(* IEC 61131-3 sources: HappyLearnCodesys/content/softmotion/CNC09_ToolLengthCorr, 3 files *)

(* ---- GVL.st ---- *)
VAR_GLOBAL CONSTANT
	gc_dwCycle : DWORD := 4000;
	gc_eOriConvention : SMC_ORI_CONVENTION := SMC_ORI_CONVENTION.ZYZ;
END_VAR

(* ---- CNC.st ---- *)
PROGRAM CNC
VAR
	iState: INT;
	pX, pY, pZ, pA: MC_Power;

	ipo: SMC_Interpolator;
	trafo: SMC_TRAFO_Gantry3;
	trafof: SMC_TRAFOF_Gantry3D;
	cabpX, cabpY, cabpZ, cabpA: SMC_ControlAxisByPos;

	tlc : SMC_ToolLengthCorr;
END_VAR

pX(
	Enable:= TRUE,
	bRegulatorOn:= TRUE,
	bDriveStart:= TRUE,
	Axis:= AxisX);
pY(
	Enable:= TRUE,
	bRegulatorOn:= TRUE,
	bDriveStart:= TRUE,
	Axis:= AxisY);
pZ(
	Enable:= TRUE,
	bRegulatorOn:= TRUE,
	bDriveStart:= TRUE,
	Axis:= AxisZ);
pA(
	Enable:= TRUE,
	bRegulatorOn:= TRUE,
	bDriveStart:= TRUE,
	Axis:= AxisA);

CASE iState OF
0:
	IF pX.Status AND pY.Status AND pZ.Status AND pA.Status THEN
		iState := 100;
	END_IF
100:
	Interpolation();
END_CASE

(* ---- CNC_PreparePath.st ---- *)
PROGRAM CNC_PreparePath
VAR_INPUT
	xStart: BOOL;
	sFileName: STRING := 'Application/CNC.cnc';
END_VAR
VAR_OUTPUT
	xStartIpo: BOOL;
	poqPath: Pointer to SMC_Outqueue;
END_VAR
VAR
	iState: INT;
	rncf2 : SMC_ReadNCFile2;
	nci : SMC_NCInterpreter;
	cv : SMC_CheckVelocities;
	aBufInterpreter : ARRAY[0..99] OF SMC_GeoInfo ;
END_VAR

poqPath := cv.poqDataOut;

CASE iState OF
0:	// idle
	IF xStart THEN
		iState := 10;
		xStartIpo := FALSE;
		rncf2(bExecute:= FALSE);
		nci(bExecute:= FALSE,sentences:= rncf2.sentences);
		cv(bExecute:= FALSE);
		xStart := FALSE;
	END_IF

10:	// start reading and processing
	rncf2(
        bExecute:= TRUE,
		sFileName:= sFileName);

	nci(
        bExecute:= TRUE,
		sentences := rncf2.sentences,
		nSizeOutQueue:= SIZEOF(aBufInterpreter),
		pbyBufferOutQueue:= ADR(aBufInterpreter),
        bEnableSyntaxChecks:= TRUE,
        eOriConv:= gc_eOriConvention);

	cv(
        bExecute:= TRUE,
		poqDataIn:= nci.poqDataOut);

	xStartIpo := TRUE;
	IF NOT cv.bBusy THEN
		iState:=0;
	END_IF
END_CASE
